Staubli VAL3: selectZone.pgx

program selectZone(num& x_nSelect[] (dimensions=1))
  local num i
  local num l_nIndex
  local num l_nMin
begin
  //
  // to save:
  // x_nBest [0] -# Traejctory
  // x_nBest [1] -# index
  // x_nBest [2] -# Type
  //
  // save the value
  //
  // use the first value
  //
  x_nSelect[0]=nHome[0]
  x_nSelect[1]=0
  x_nSelect[2]=nCoeff[0]
end
